(* IEC 61131-3 sources: lc3-wifi-kurs/src/example_7_Double_Click, 3 files *)

(* ---- Double_Click_In.iecfbd ---- *)
FUNCTION_BLOCK Double_Click_In
  {
    height := 80;
    width := 200;
  }

  VAR
    i2c_handle : DINT := -1;
    input_values : ARRAY[0..7] OF BOOL;
  END_VAR
  VAR_OUTPUT
    digital_in : ARRAY[0..7] OF BOOL;
  END_VAR

  (*

    // Network 1:
    LT(IN1 := i2c_handle, IN2 := 0, LT => @C(11).LT);
    I2C_open(EN := @C(11).LT, bus_id := 1, I2C_open => i2c_handle);

    // Network 2:
    @VF(9) := I2C_ADDRESSES#PCF8574_INPUT_1;
    GE(IN1 := i2c_handle, IN2 := 0, GE => @C(13).GE);
    I2C_PCF8574_read(EN := @C(13).GE, fd := i2c_handle, address := @VF(9), I2C_PCF8574_read => digital_in);

  *)

  @VF(3) : @E(i2c_handle), @R(154.3, 150.0, 140.0, 19.0);
  @VF(4) : @E(0), @R(154.3, 170.0, 140.0, 19.0), DINT;
  @VF(5) : @E(1), @R(150.0, 192.5, 140.0, 19.0), INT;
  @VF(6) : @E(0), @R(153.5, 283.5, 140.0, 19.0), DINT;
  @VF(7) : @E(i2c_handle), @R(153.5, 303.5, 140.0, 19.0);
  @VF(8) : @E(i2c_handle), @R(807.6, 187.9, 140.0, 19.0);
  @VF(9) : @E(I2C_ADDRESSES#PCF8574_INPUT_1), @R(153.5, 323.5, 140.0, 19.0);
  @C(11) : @F(LT), @R(334.3, 150.0, 40.0, 38.0), DINT, @I(@N(IN1), @L(9.5)), @I(@N(IN2), @L(29.5)), @O(@N(LT), @R(9.5));
  @C(12) : @F(I2C_open), @R(547.6, 167.9, 160.0, 38.5), @I(@N(EN), @L(9.5)), @I(@N(bus_id), @L(29.5)), @O(@N(ENO), @R(9.5)), @O(@N(I2C_open), @R(29.5));
  @C(13) : @F(GE), @R(380.7, 257.8, 40.0, 38.0), DINT, @I(@N(IN1), @L(9.5)), @I(@N(IN2), @L(29.5)), @O(@N(GE), @R(9.5));
  @C(14) : @F(I2C_PCF8574_read), @R(552.0, 284.7, 160.0, 58.0), @I(@N(EN), @L(9.5)), @I(@N(fd), @L(29.5)), @I(@N(address), @L(49.5)), @O(@N(ENO), @R(9.5)), @O(@N(I2C_PCF8574_read), @R(29.5));
  @VF(2) : @E(digital_in), @R(816.0, 304.5, 140.0, 19.0);
  @CP(15) : 333.6, 313.0;

  @G(16) :
     @L(@VF(3).o, @C(11).IN1)
    ;
  @G(17) :
     @L(@VF(4).o, @C(11).IN2)
    ;
  @G(18) :
     @L(@C(11).LT, @C(12).EN)
    ;
  @G(19) :
     @L(@VF(5).o, @C(12).bus_id)
    ;
  @G(20) :
     @L(@C(13).GE, @C(14).EN)
    ;
  @G(21) :
     @L(@VF(6).o, @C(13).IN2)
    ;
  @G(22) :
     @L(@VF(7).o, @CP(15)),
     @L(@CP(15), @C(14).fd),
     @L(@CP(15), @C(13).IN1)
    ;
  @G(23) :
     @L(@C(12).I2C_open, @VF(8).i)
    ;
  @G(24) :
     @L(@VF(9).o, @C(14).address)
    ;
  @G(10) :
     @L(@C(14).I2C_PCF8574_read, @VF(2).i)
    ;
END_FUNCTION_BLOCK

(* ---- Double_Click_Out.iecfbd ---- *)
FUNCTION_BLOCK Double_Click_Out
  {
    height := 80;
    width := 200;
  }

  VAR
    i2c_handle : DINT := -1;
    input_values : ARRAY[0..7] OF BOOL;
  END_VAR
  VAR_INPUT
    digital_out : ARRAY[0..7] OF BOOL;
  END_VAR

  (*

    // Network 1:
    LT(IN1 := i2c_handle, IN2 := 0, LT => @C(11).LT);
    I2C_open(EN := @C(11).LT, bus_id := 1, I2C_open => i2c_handle);

    // Network 2:
    @VF(28) := I2C_ADDRESSES#PCF8574_OUTPUT_1;
    GE(IN1 := i2c_handle, IN2 := 0, GE => @C(30).GE);
    I2C_PCF8574_write(EN := @C(30).GE, fd := i2c_handle, address := @VF(28), pin_values := digital_out);

  *)

  @VF(3) : @E(i2c_handle), @R(154.3, 150.0, 140.0, 19.0);
  @VF(4) : @E(0), @R(154.3, 170.0, 140.0, 19.0), DINT;
  @VF(5) : @E(1), @R(150.0, 192.5, 140.0, 19.0), INT;
  @VF(8) : @E(i2c_handle), @R(807.6, 187.9, 140.0, 19.0);
  @C(11) : @F(LT), @R(334.3, 150.0, 40.0, 38.0), DINT, @I(@N(IN1), @L(9.5)), @I(@N(IN2), @L(29.5)), @O(@N(LT), @R(9.5));
  @C(12) : @F(I2C_open), @R(547.6, 167.9, 160.0, 38.5), @I(@N(EN), @L(9.5)), @I(@N(bus_id), @L(29.5)), @O(@N(ENO), @R(9.5)), @O(@N(I2C_open), @R(29.5));
  @VF(1) : @E(digital_out), @R(153.6, 354.5, 140.0, 19.0);
  @VF(26) : @E(i2c_handle), @R(153.6, 314.5, 140.0, 19.0);
  @VF(27) : @E(0), @R(153.6, 294.5, 140.0, 19.0), DINT;
  @VF(28) : @E(I2C_ADDRESSES#PCF8574_OUTPUT_1), @R(153.6, 334.5, 140.0, 19.0);
  @C(30) : @F(GE), @R(483.6, 274.5, 40.0, 38.0), DINT, @I(@N(IN1), @L(9.5)), @I(@N(IN2), @L(29.5)), @O(@N(GE), @R(9.5));
  @C(31) : @F(I2C_PCF8574_write), @R(618.0, 288.0, 160.0, 88.0), @I(@N(EN), @L(19.5)), @I(@N(fd), @L(39.5)), @I(@N(address), @L(59.5)), @I(@N(pin_values), @L(79.5)), @O(@N(ENO), @R(19.5));
  @CP(32) : 371.4, 324.0;

  @G(16) :
     @L(@VF(3).o, @C(11).IN1)
    ;
  @G(17) :
     @L(@VF(4).o, @C(11).IN2)
    ;
  @G(18) :
     @L(@C(11).LT, @C(12).EN)
    ;
  @G(19) :
     @L(@VF(5).o, @C(12).bus_id)
    ;
  @G(23) :
     @L(@C(12).I2C_open, @VF(8).i)
    ;
  @G(33) :
     @L(@VF(26).o, @CP(32)),
     @L(@CP(32), @C(31).fd),
     @L(@CP(32), @C(30).IN1)
    ;
  @G(34) :
     @L(@VF(27).o, @C(30).IN2)
    ;
  @G(35) :
     @L(@VF(28).o, @C(31).address)
    ;
  @G(36) :
     @L(@C(30).GE, @C(31).EN)
    ;
  @G(25) :
     @L(@VF(1).o, @C(31).pin_values)
    ;
END_FUNCTION_BLOCK

(* ---- Program_Double_Click.iecfbd ---- *)
PROGRAM Program_Double_Click
  VAR
    digital_in : ARRAY[0..7] OF BOOL;
    digital_out : ARRAY[0..7] OF BOOL;
    Double_Click_In1 : Double_Click_In;
    Double_Click_Out1 : Double_Click_Out;
    Multi_Click1 : Multi_Click;
  END_VAR

  (*

    // Network 1:
    Double_Click_In1();
    digital_in := Double_Click_In1.digital_in;

    // Network 2:
    Multi_Click1(in := digital_in[0], period := T#500ms, CV := 2);
    Toggle(in := Multi_Click1.out, value := digital_out[0], out => digital_out[0]);

    // Network 3:
    Double_Click_Out1(digital_out := digital_out);

  *)

  @C(1) : @FB(Double_Click_In1), @R(200.0, 200.0, 200.0, 80.0), @O(@N(digital_in), @R(9.5));
  @C(2) : @FB(Double_Click_Out1), @R(420.0, 510.0, 200.0, 80.0), @I(@N(digital_out), @L(9.5));
  @VF(3) : @E(digital_in), @R(420.0, 200.0, 140.0, 19.0);
  @VF(5) : @E(digital_out), @R(147.0, 512.3, 140.0, 19.0);
  @VF(8) : @E(digital_in[0]), @R(210.0, 350.0, 140.0, 19.0);
  @VF(9) : @E(digital_out[0]), @R(930.0, 350.0, 140.0, 19.0);
  @VF(10) : @E(T#500ms), @R(210.0, 370.0, 140.0, 19.0);
  @VF(14) : @E(digital_out[0]), @R(580.0, 370.0, 140.0, 19.0);
  @VF(22) : @E(2), @R(210.0, 390.0, 140.0, 19.0), INT;
  @C(7) : @FB(Multi_Click1), @R(440.0, 350.0, 120.0, 130.0), @I(@N(in), @L(9.5)), @I(@N(period), @L(29.5)), @I(@N(CV), @L(49.5)), @O(@N(out), @R(9.5));
  @C(13) : @F(Toggle), @R(760.0, 350.0, 120.0, 38.0), @I(@N(in), @L(9.5)), @I(@N(value), @L(29.5)), @O(@N(out), @R(9.5));

  @G(4) :
     @L(@C(1).digital_in, @VF(3).i)
    ;
  @G(6) :
     @L(@VF(5).o, @C(2).digital_out)
    ;
  @G(11) :
     @L(@VF(8).o, @C(7).in)
    ;
  @G(12) :
     @L(@VF(10).o, @C(7).period)
    ;
  @G(20) :
     @L(@VF(22).o, @C(7).CV)
    ;
  @G(15) :
     @L(@C(7).out, @C(13).in)
    ;
  @G(16) :
     @L(@VF(14).o, @C(13).value)
    ;
  @G(17) :
     @L(@C(13).out, @VF(9).i)
    ;
END_PROGRAM
